(* IEC 61131-3 sources: ICSQuartz/benchmarks/oscat_basic_trim1/src, 1 file *)

(* ---- program.st ---- *)
PROGRAM PLC_PRG
VAR_INPUT
    in_STR: STRING;
END_VAR

TRIM1(in_STR);

END_PROGRAM
